// TIA Portal V18 export
DATA_BLOCK "CoordinationHmi"   // DB1
{ S7_Optimized_Access := 'FALSE' }
// stored: AutoNumber false
   VAR
      CoordinationConsoleHmi : Array[0..15] of Bool;
      CoordinationHpuHmi : Array[0..15] of Bool;
      CoordinationDoghouseHmi : Array[0..15] of Bool;
      RTClock : DTL;
   END_VAR
BEGIN
END_DATA_BLOCK
